Staubli VAL3: Control_PanelMd.pgx

public program Control_PanelMd(string x_sMess)
begin

  call Control_PanelS("",2,3,34,4)
  call Control_ListCls()
  x_sMess=left(x_sMess,min(getDisplayLen(x_sMess),nPanelWidthX))
  gotoxy(nPanelLTopX+ (nPanelWidthX-getDisplayLen(x_sMess))/2,nPanelLTopY+nPanelLengthY/2+1)
  put( x_sMess)


end
